# EPICS substitutions: KS3497xAApp/Db/KS3497xA_channels.substitutions
# File: KS3497xA_channels.substitutions
# Author: Wayne Lewis <wlewis@lbl.gov>
# Date: 2019-09-16
#
# Description:
# Substitutions file to load database for multiple channels
#
# Revisions:
#
# Copyright:
# Lawrence Berkeley National Laboratory
#
# Licence:
# TBD

file "KS3497xA_channel.template" {
pattern	{"C"}
		{"101"}
		{"102"}
		{"103"}
		{"104"}
		{"105"}
		{"106"}
		{"107"}
		{"108"}
		{"109"}
		{"110"}
		{"111"}
		{"112"}
		{"113"}
		{"114"}
		{"115"}
		{"116"}
}
